PROGRAM MAIN
VAR
END_VAR

END_PROGRAM

(* stored: Version 1.1.0.1
   POU MAIN: Id {53223da0-e4c3-44d1-98c8-c51b0f8ea35c} *)
